FUNCTION_BLOCK EnumeratorBase
VAR
	connection : EnumeratorConnection;
END_VAR

METHOD PUBLIC Dispose
VAR_INPUT
END_VAR
connection.Dispose();
END_METHOD

METHOD FB_init : BOOL
VAR_INPUT
	bInitRetains : BOOL; // if TRUE, the retain variables are initialized (warm start / cold start)
	bInCopyCode : BOOL;  // if TRUE, the instance afterwards gets moved into the copy code (online change)
	ConnectionUpdater : I_EnumeratorConnectionUpdater;
END_VAR
connection.LinkTo(ConnectionUpdater);
END_METHOD

PROPERTY PUBLIC IsValid : BOOL
GET
IsValid := connection.IsValid;
END_GET
END_PROPERTY

END_FUNCTION_BLOCK

(* stored: Version 1.1.0.1, ProductVersion 3.1.4024.12
   POU EnumeratorBase: Id {ab0e0f95-5b7e-4770-acc0-5bd568950a14}, SpecialFunc None
   Folder Constructor: Id {d796c509-27ba-4f7b-abac-cf86cee01e7f}
   Method Dispose: Id {c0409b25-95a3-4fca-8e23-1f146ce9444c}
   Method FB_init: Id {db5c1070-779b-4e22-a925-e7b14274daf2}
   Property IsValid: Id {971570d5-4dee-430c-9e4a-5d200224b7cc}
   Get Get: Id {801958b5-4378-4c4e-a9c2-65873e5184a8} *)
